TYPE ST_IpStackDiagSub :
	STRUCT
		nSendCnt : UDINT;
		nSendFailCnt : UDINT;
		nRecvCnt : UDINT;
		nRecvFailCnt : UDINT;
	END_STRUCT
END_TYPE

(* stored: Version 1.1.0.1, ProductVersion 3.1.4024.13
   DUT ST_IpStackDiagSub: Id {c11b0ac8-58a7-4342-98cd-c3532577edd7} *)
